TYPE ST_AlarmLog :
STRUCT
	sTimestamp: STRING;
	sText: STRING(255); //
	sSourceName: STRING(255); //
	EventClassName: STRING(255); //
    eConfirmationState : INT;
    eSeverity :  INT; // INT
END_STRUCT
END_TYPE

(* stored: Version 1.1.0.1, ProductVersion 3.1.4026.18
   DUT ST_AlarmLog: Id {b4939509-00b7-445d-8704-756932ed98ff} *)
